{attribute 'GeneratedUsingTerminal: EL6731--0000'}
{attribute addProperty BoxType "EL6731--0000"}
{attribute addProperty Id "EtcSlaveTerminalBaseInfoDataAT %I*InfoData_90184F0C16"}
{attribute addProperty CRC "354618671"}
{attribute addProperty Size "16"}
TYPE EL6731_15230D2F EXTENDS EtcSlaveTerminalBase :
STRUCT
	{attribute addProperty Name "InfoData"}
	InfoData : InfoData_90184F0C;
END_STRUCT
END_TYPE

(* stored: Version 1.2.0.0, ProductVersion 3.1.4024.9
   DUT EL6731_15230D2F: Id {cf7fbd37-e12a-4996-b149-f5f722d755ae} *)
